TYPE ST_SIZE :
STRUCT
	nValue : UDINT;
END_STRUCT
END_TYPE

(* stored: Version 1.1.0.1, ProductVersion 3.1.4024.15
   DUT ST_SIZE: Id {a0e6c432-dffd-4b82-97f4-945f45effaa9} *)
